FUNCTION Disable_System : INT

VAR_IN_OUT
	RGP: System;
END_VAR

VAR

	CR1278_TOOL_OUTRIGGER_RET: INT;
END_VAR

//Disables the Movment Axes
	Disable_Axis(RGP.EN1000.DV1150_TRANSX_DRIVE);
	Disable_Axis(RGP.EN1000.DV1175_TRANSY_DRIVE);
	Disable_Axis(RGP.EN1000.DV1325_POS_TOOL_ROTZ_DRIVE);
	Disable_Axis(RGP.EN1000.DV1151_JACK1_DRIVE);
	Disable_Axis(RGP.EN1000.DV1275_JACK2_DRIVE);
	Disable_Axis(RGP.EN1000.DV1301_JACK3_DRIVE);
	Disable_Axis(RGP.EN1000.RIO1135_MON_TOOL_ROTZ_DRIVE);
	
//Program Variables
	// Axis Enable booleans
	RGP.PROG.TRANSX_POS_EN := 0;
	RGP.PROG.TRANSX_NEG_EN := 0;
	RGP.PROG.TRANSY_POS_EN := 0;
	RGP.PROG.TRANSY_NEG_EN := 0;
	RGP.PROG.POS_TOOL_ROTZ_POS_EN := 0;
	RGP.PROG.POS_TOOL_ROTZ_NEG_EN := 0;	
	RGP.PROG.JACK1_POS_EN := 0;
	RGP.PROG.JACK1_NEG_EN := 0;
	RGP.PROG.JACK2_POS_EN := 0;
	RGP.PROG.JACK2_NEG_EN := 0;
	RGP.PROG.JACK3_POS_EN := 0;
	RGP.PROG.JACK3_NEG_EN := 0;
	RGP.PROG.MON_TOOL_ROTZ_POS_EN := 0;
	RGP.PROG.MON_TOOL_ROTZ_NEG_EN := 0;
	
	// Axis Speeds
	RGP.PROG.TRANSX_SPEED := 0;
	RGP.PROG.TRANSY_SPEED := 0;
	RGP.PROG.POS_TOOL_ROTZ_SPEED := 0;
	RGP.PROG.All_JACKS_SPEED := 0; 
	RGP.PROG.JACK1_SPEED := 0;
	RGP.PROG.JACK2_SPEED := 0;
	RGP.PROG.JACK3_SPEED := 0;
	RGP.PROG.MON_TOOL_ROTZ_SPEED := 0;

END_FUNCTION

(* stored: Version 1.1.0.1, ProductVersion 3.1.4024.0
   POU Disable_System: Id {6ed0d971-90d8-41aa-828d-e5e64729759f}, SpecialFunc None *)
